SUBAPPLICATION func (* Subapplication Type *)
  (* Standard: 61499-2 *)
  (* Version 1.0, 2023-02-17, Franz *)
  IMPORT DefaultPool::Button_Reset_Gesamtzaehler;
  IMPORT DefaultPool::Button_Reset_Tageszaehler;
  IMPORT DefaultPool::NumberVariable_Gesamtzaehler;
  IMPORT DefaultPool::NumberVariable_Gesamtziel;
  IMPORT DefaultPool::NumberVariable_Tageszaehler;
  IMPORT DefaultPool::NumberVariable_Tagesziel;
  IMPORT DefaultPool::ObjectPointer_Gesamtziel;
  IMPORT DefaultPool::ObjectPointer_Tagesziel;
  IMPORT DefaultPool::SoftKey_Reset_Gesamtzaehler;
  IMPORT DefaultPool::SoftKey_Reset_Tageszaehler;
  IMPORT NVS_Keys::KEY_GESAMTZAEHLER;
  IMPORT NVS_Keys::KEY_GESAMTZIEL;
  IMPORT NVS_Keys::KEY_TAGESZAEHLER;
  IMPORT NVS_Keys::KEY_TAGESZIEL;
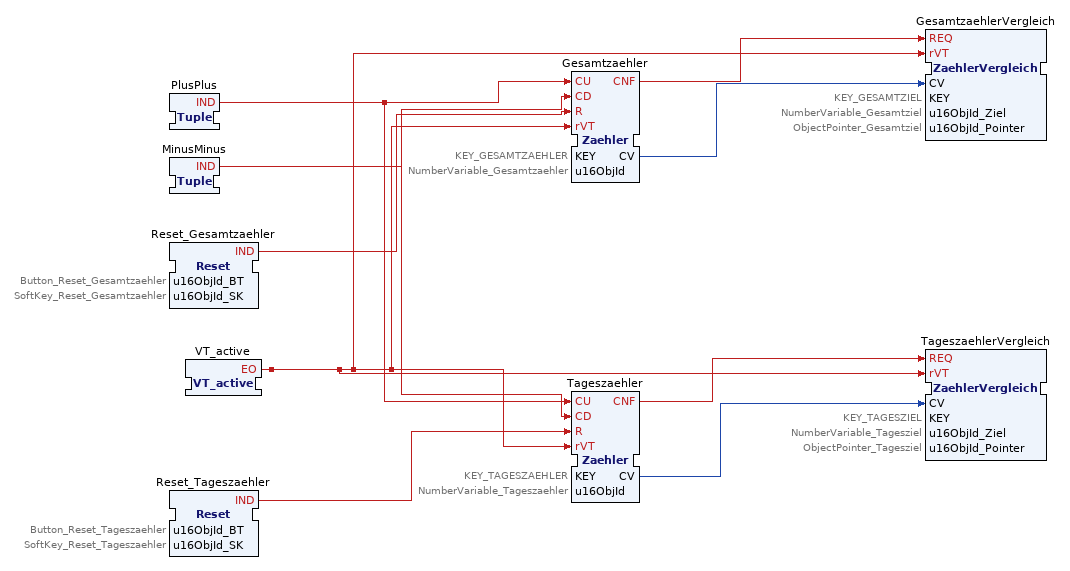
  SUBAPPS
    VT_active : VT_active;
    MinusMinus : Tuple;
    PlusPlus : Tuple;
    Reset_Gesamtzaehler : Reset(u16ObjId_BT := Button_Reset_Gesamtzaehler, u16ObjId_SK := SoftKey_Reset_Gesamtzaehler);
    Reset_Tageszaehler : Reset(u16ObjId_BT := Button_Reset_Tageszaehler, u16ObjId_SK := SoftKey_Reset_Tageszaehler);
    Gesamtzaehler : Zaehler(KEY := KEY_GESAMTZAEHLER, u16ObjId := NumberVariable_Gesamtzaehler);
    Tageszaehler : Zaehler(KEY := KEY_TAGESZAEHLER, u16ObjId := NumberVariable_Tageszaehler);
    TageszaehlerVergleich : ZaehlerVergleich(KEY := KEY_TAGESZIEL, u16ObjId_Ziel := NumberVariable_Tagesziel, u16ObjId_Pointer := ObjectPointer_Tagesziel);
    GesamtzaehlerVergleich : ZaehlerVergleich(KEY := KEY_GESAMTZIEL, u16ObjId_Ziel := NumberVariable_Gesamtziel, u16ObjId_Pointer := ObjectPointer_Gesamtziel);
  END_SUBAPPS
  EVENT_CONNECTIONS
    PlusPlus.IND TO Gesamtzaehler.CU;
    MinusMinus.IND TO Gesamtzaehler.CD;
    Reset_Gesamtzaehler.IND TO Gesamtzaehler.R;
    VT_active.EO TO Gesamtzaehler.rVT;
    PlusPlus.IND TO Tageszaehler.CU;
    MinusMinus.IND TO Tageszaehler.CD;
    Reset_Tageszaehler.IND TO Tageszaehler.R;
    VT_active.EO TO Tageszaehler.rVT;
    Tageszaehler.CNF TO TageszaehlerVergleich.REQ;
    VT_active.EO TO TageszaehlerVergleich.rVT;
    Gesamtzaehler.CNF TO GesamtzaehlerVergleich.REQ;
    VT_active.EO TO GesamtzaehlerVergleich.rVT;
  END_CONNECTIONS
  DATA_CONNECTIONS
    Tageszaehler.CV TO TageszaehlerVergleich.CV;
    Gesamtzaehler.CV TO GesamtzaehlerVergleich.CV;
  END_CONNECTIONS
END_SUBAPPLICATION
